{attribute 'qualified_only'}
VAR_GLOBAL CONSTANT
	SerializerMaxColumns : INT := 10;
	DeserializerMaxColumns : INT := 10;
END_VAR

(* stored: Version 1.1.0.1
   GVL TableSerializationParameters: Id {18fa224f-895c-08b7-0652-17bfee0d9dec}, ParameterList True *)
